PROGRAM MAIN
VAR
END_VAR

Prg_FSM();

END_PROGRAM

(* stored: Version 1.1.0.1, ProductVersion 3.1.4024.9
   POU MAIN: Id {f7c03209-2fcf-45de-b609-0efb1efda840}, SpecialFunc None *)
